# EPICS substitutions: NucInstDigApp/Db/NucInstDigDCSpec.substitutions
global { "P=\$(P)", "Q=\$(Q)" }

file "NucInstDigDCSpec.template" {
    pattern { N }
    { "1" }
    { "2" }
    { "3" }
    { "4" }
}
